TYPE TcaPushButtonService :
STRUCT
	Button : BOOL;
	Light : BOOL;	
END_STRUCT
END_TYPE

(* stored: Version 1.1.0.1
   DUT TcaPushButtonService: Id {08f25f94-4b94-479f-a8ca-32cbd1ebeec1} *)
